TYPE ST_FireDetection_get :
STRUCT
	b_FireAlarm		: 	BOOL;
	SmokeDetectors 	:	ST_SmokeDetectors;
	CODetectors		:	ST_CODetectors;
	Events			:	ST_FireSystem_Events;
END_STRUCT
END_TYPE

(* stored: Version 1.1.0.1, ProductVersion 3.1.4026.18
   DUT ST_FireDetection_get: Id {6cc78167-32bf-4519-8037-010d2b675e1a} *)
